% RSLogix 500 project ComprobarActuadoresSensores.RSS, saved by version 8.30.00.15 %
PROJECT "UNTITLED"    % processor: Bul.1763 MicroLogix 1100 Series B %

PROGRAM FILES
  LAD 2   12 rungs
  LAD 3 "PID"  4 rungs

DATA FILES
  O0 OUTPUT  6 elements
  I1 INPUT  12 elements
  S2 STATUS  66 elements
  B3 BINARY  1 elements
  T4 TIMER  1 elements
  C5 COUNTER  1 elements
  R6 CONTROL  1 elements
  N7 INTEGER  4 elements
  F8 FLOAT  3 elements
  PD9   1 elements
  N10   11 elements
  N11   1 elements
  N12   1 elements
  PD22   10 elements

LADDER 2
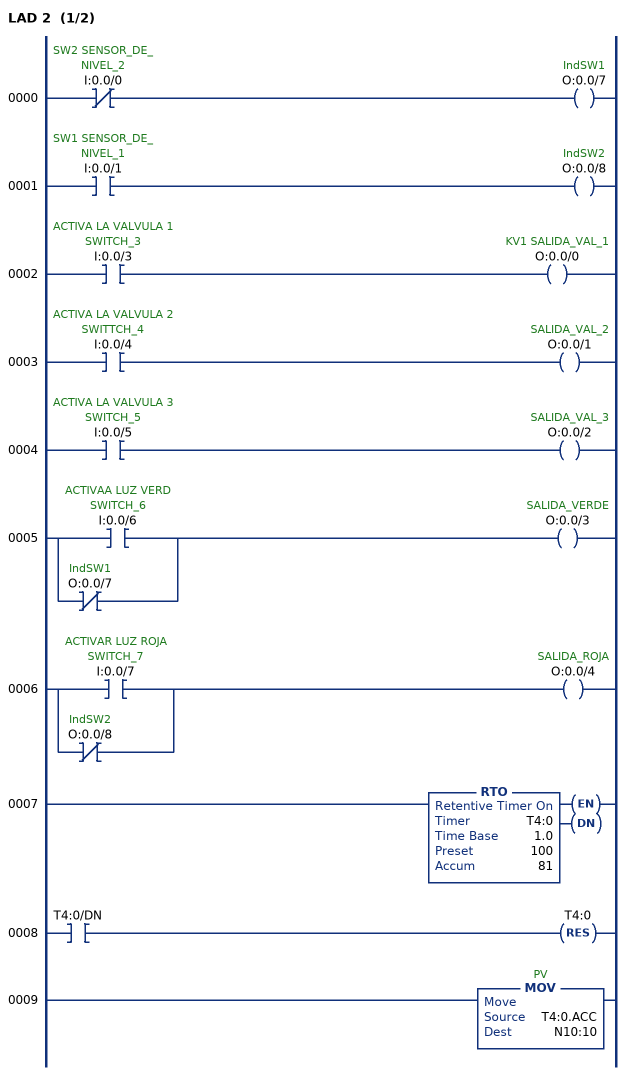
% Rung: 0 %
SOR XIO I:0.0/0 OTE O:0.0/7 EOR
%   I:0.0/0  SENSOR_DE_NIVEL_2  "SW2" %
%   O:0.0/7  "IndSW1" %
% Rung: 1 %
SOR XIC I:0.0/1 OTE O:0.0/8 EOR
%   I:0.0/1  SENSOR_DE_NIVEL_1  "SW1" %
%   O:0.0/8  "IndSW2" %
% Rung: 2 %
SOR XIC I:0.0/3 OTE O:0.0/0 EOR
%   I:0.0/3  SWITCH_3  "ACTIVA LA VALVULA 1" %
%   O:0.0/0  SALIDA_VAL_1  "KV1" %
% Rung: 3 %
SOR XIC I:0.0/4 OTE O:0.0/1 EOR
%   I:0.0/4  SWITTCH_4  "ACTIVA LA VALVULA 2" %
%   O:0.0/1  SALIDA_VAL_2 %
% Rung: 4 %
SOR XIC I:0.0/5 OTE O:0.0/2 EOR
%   I:0.0/5  SWITCH_5  "ACTIVA LA VALVULA 3" %
%   O:0.0/2  SALIDA_VAL_3 %
% Rung: 5 %
SOR BST XIC I:0.0/6 NXB XIO O:0.0/7 BND OTE O:0.0/3 EOR
%   I:0.0/6  SWITCH_6  "ACTIVAA LUZ VERD" %
%   O:0.0/7  "IndSW1" %
%   O:0.0/3  SALIDA_VERDE %
% Rung: 6 %
SOR BST XIC I:0.0/7 NXB XIO O:0.0/8 BND OTE O:0.0/4 EOR
%   I:0.0/7  SWITCH_7  "ACTIVAR LUZ ROJA" %
%   O:0.0/8  "IndSW2" %
%   O:0.0/4  SALIDA_ROJA %
% Rung: 7 %
SOR RTO T4:0 1.0 100 81 EOR
% Rung: 8 %
SOR XIC T4:0/DN RES T4:0 EOR
% Rung: 9 %
SOR MOV T4:0.ACC N10:10 EOR
%   N10:10  "PV" %

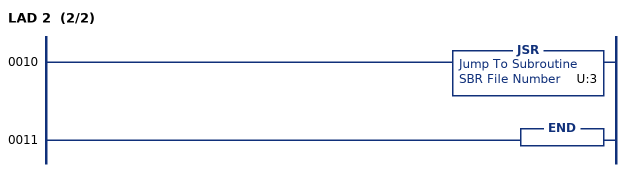
% Rung: 10 %
SOR JSR U:3 EOR
% Rung: 11 %
SOR END EOR

LADDER 3 "PID"
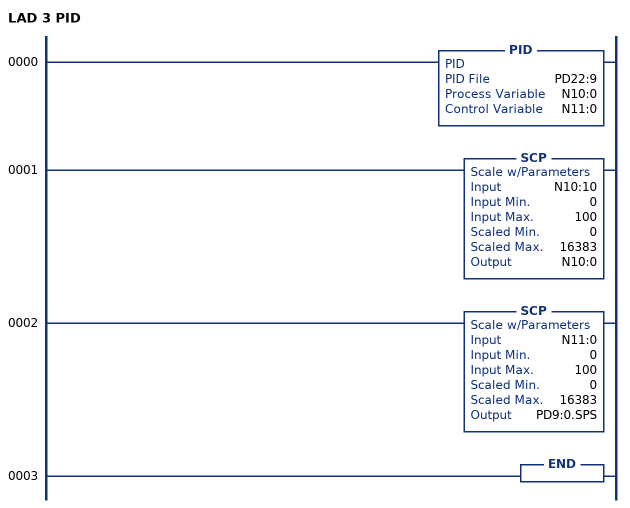
% Rung: 0 %
SOR PID PD22:9 N10:0 N11:0 EOR
% Rung: 1 %
SOR SCP N10:10 0 100 0 16383 N10:0 EOR
%   N10:10  "PV" %
% Rung: 2 %
SOR SCP N11:0 0 100 0 16383 PD9:0.SPS EOR
% Rung: 3 %
SOR END EOR

OTHER DOCUMENTED ADDRESSES
  O:0.0/6  "ENCLAVE"

DATA TABLE (non-zero values as saved)
DATA T4
% .PRE .ACC %
% T4:0 % 100 81
DATA N7
% N7:0 % 20 20 0 1638
DATA F8
% F8:0 % 0 200 1.080757
DATA N10
% N10:0 % 13434 0 0 0 0 0 0 0 0 0
% N10:10 % 82
DATA N11
% N11:0 % 2457
DATA N12
% N12:0 % 20
